{attribute addProperty BoxType "EJ1957-0000-0017"}
{attribute addProperty Id "FSOEAT %I*FSOE_085426AE567"}
{attribute addProperty CRC "3826593544"}
{attribute addProperty SizeInBites "56"}
{attribute addProperty SizeInBytes "7"}
TYPE FSoE_Inputs_E4152F08 :
STRUCT
	{attribute addProperty Name "FSOE"}
	FSOE AT %I* : FSOE_085426AE;
END_STRUCT
END_TYPE

(* stored: Version 1.2.0.0, ProductVersion 3.1.4024.9
   DUT FSoE_Inputs_E4152F08: Id {40f60b1a-2004-4aa3-b4e1-6859259eb75b} *)
